// TIA Portal project "ExamenTIA" (V15)

(* hardware
DEVICE "S7-1200 station_1"  S7-1200 Station
   slot 0: "Rack_0"  S7-1200 Rack  Rack  V1.0
   slot 1: "PLC_1"  CPU 1214C AC/DC/Rly  6ES7 214-1BG40-0XB0  V4.2
*)

// ===== PLC "PLC_1"  CPU 1214C AC/DC/Rly =====

VAR_GLOBAL   // PLC tag table "Tabla de variables estándar"
   "Clock_Byte" AT %MB0 : Byte;
   "Clock_10Hz" AT %M0.0 : Bool;
   "Clock_5Hz" AT %M0.1 : Bool;
   "Clock_2.5Hz" AT %M0.2 : Bool;
   "Clock_2Hz" AT %M0.3 : Bool;
   "Clock_1.25Hz" AT %M0.4 : Bool;
   "Clock_1Hz" AT %M0.5 : Bool;
   "Clock_0.625Hz" AT %M0.6 : Bool;
   "Clock_0.5Hz" AT %M0.7 : Bool;
   "S_Abajo" AT %I0.0 : Bool;
   "S_Arriba" AT %I0.1 : Bool;
   "S_Peso" AT %I0.2 : Bool;
   "Seta" AT %I0.3 : Bool;
   "Auto" AT %I0.4 : Bool;
   "Manu" AT %I0.5 : Bool;
   "M_Alante" AT %I0.6 : Bool;
   "M_Atras" AT %I0.7 : Bool;
   "Paro" AT %I1.0 : Bool;
   "Rearme" AT %I1.1 : Bool;
   "Motor_Alante" AT %Q0.0 : Bool;
   "Motor_Atras" AT %Q0.1 : Bool;
   "L_Alante" AT %Q0.2 : Bool;
   "L_Paro" AT %Q0.3 : Bool;
   "L_ParoE" AT %Q0.4 : Bool;
   "L_Atras" AT %Q0.5 : Bool;
   "L_Sobrecarga" AT %Q0.6 : Bool;
   "FlancoP" AT %M10.0 : Bool;
   "Aux_seta" AT %M10.1 : Bool;
   "Aux_sobrecarga" AT %M10.2 : Bool;
   "FlancoN" AT %M10.3 : Bool;
   "Aux1" AT %M10.4 : Bool;
END_VAR

// folder: System blocks/Program resources

DATA_BLOCK "IEC_Timer_0_DB"   // DB1
{ S7_Optimized_Access := 'TRUE' }
AUTHOR : Simatic
FAMILY : IEC
NAME : IEC_TMR
VERSION : 1.0
// stored: InstanceOfName IEC_TIMER
"IEC_TIMER"
BEGIN
END_DATA_BLOCK

// folder: (top level)

FUNCTION "Automático" : Void   // FC1, LAD
{ S7_Optimized_Access := 'TRUE' }
VERSION : 0.1
   VAR_TEMP   // added for the SCL form of the ladder/FBD networks
      _w1 : Bool;
   END_VAR
BEGIN

REGION Network 1
   // Cuando el sensor de abajo detecta a peso activa la rampa y reinicia el temporizador de paro
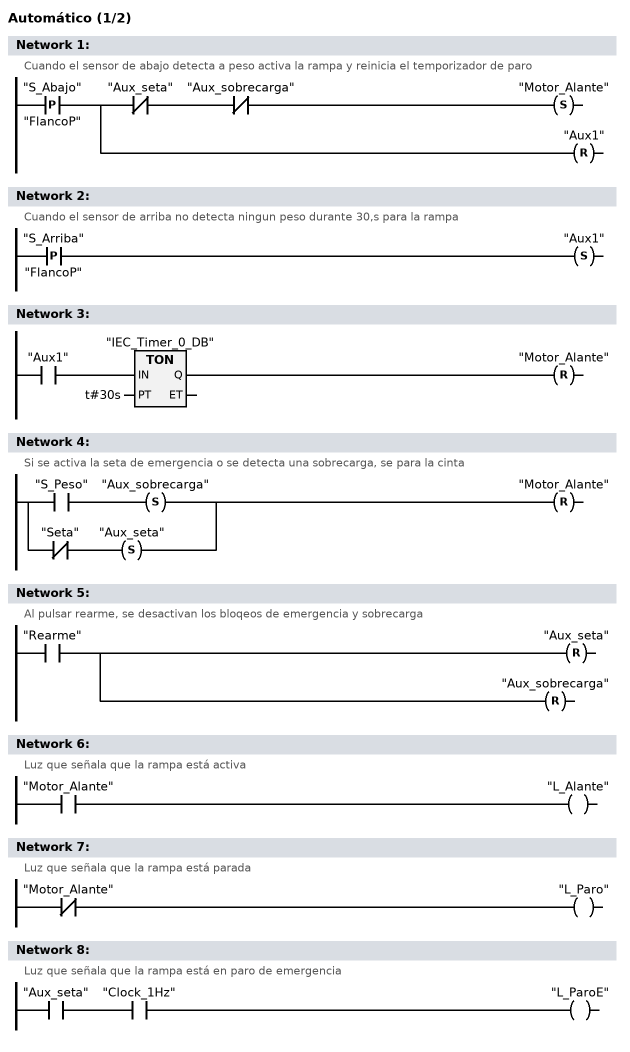
   RUNG wire#powerrail
      P_Contact(operand := "S_Abajo", bit := "FlancoP")
      wire#w1
      I_Contact( "Aux_seta" )
      I_Contact( "Aux_sobrecarga" )
      S_Coil( "Motor_Alante" )
   END_RUNG
   RUNG wire#w1
      R_Coil( "Aux1" )
   END_RUNG
   // the same network as SCL:
   #_w1 := "S_Abajo" AND NOT "FlancoP";   // rising edge of "S_Abajo"
   "FlancoP" := "S_Abajo";
   IF #_w1 AND NOT "Aux_seta" AND NOT "Aux_sobrecarga" THEN "Motor_Alante" := TRUE; END_IF;
   IF #_w1 THEN "Aux1" := FALSE; END_IF;
END_REGION

REGION Network 2
   // Cuando el sensor de arriba no detecta ningun peso durante 30,s para la rampa
   RUNG wire#powerrail
      P_Contact(operand := "S_Arriba", bit := "FlancoP")
      S_Coil( "Aux1" )
   END_RUNG
   // the same network as SCL:
   #_w1 := "S_Arriba" AND NOT "FlancoP";   // rising edge of "S_Arriba"
   "FlancoP" := "S_Arriba";
   IF #_w1 THEN "Aux1" := TRUE; END_IF;
END_REGION

REGION Network 3
   "IEC_Timer_0_DB".TON(IN := "Aux1", PT := t#30s);
   IF "IEC_Timer_0_DB".Q THEN "Motor_Alante" := FALSE; END_IF;
END_REGION

REGION Network 4
   // Si se activa la seta de emergencia o se detecta una sobrecarga, se para la cinta
   RUNG wire#powerrail
      Contact( "S_Peso" )
      S_Coil( "Aux_sobrecarga" )
      wire#w1
      R_Coil( "Motor_Alante" )
   END_RUNG
   RUNG wire#powerrail
      I_Contact( "Seta" )
      S_Coil( "Aux_seta" )
   END_RUNG wire#w1
   // the same network as SCL:
   IF "S_Peso" THEN "Aux_sobrecarga" := TRUE; END_IF;
   IF NOT "Seta" THEN "Aux_seta" := TRUE; END_IF;
   IF "S_Peso" OR NOT "Seta" THEN "Motor_Alante" := FALSE; END_IF;
END_REGION

REGION Network 5
   // Al pulsar rearme, se desactivan los bloqeos de emergencia y sobrecarga
   RUNG wire#powerrail
      Contact( "Rearme" )
      wire#w1
      R_Coil( "Aux_seta" )
   END_RUNG
   RUNG wire#w1
      R_Coil( "Aux_sobrecarga" )
   END_RUNG
   // the same network as SCL:
   IF "Rearme" THEN
       "Aux_seta" := FALSE;
       "Aux_sobrecarga" := FALSE;
   END_IF;
END_REGION

REGION Network 6
   // Luz que señala que la rampa está activa
   RUNG wire#powerrail
      Contact( "Motor_Alante" )
      Coil( "L_Alante" )
   END_RUNG
   // the same network as SCL:
   "L_Alante" := "Motor_Alante";
END_REGION

REGION Network 7
   // Luz que señala que la rampa está parada
   RUNG wire#powerrail
      I_Contact( "Motor_Alante" )
      Coil( "L_Paro" )
   END_RUNG
   // the same network as SCL:
   "L_Paro" := NOT "Motor_Alante";
END_REGION

REGION Network 8
   // Luz que señala que la rampa está en paro de emergencia
   RUNG wire#powerrail
      Contact( "Aux_seta" )
      Contact( "Clock_1Hz" )
      Coil( "L_ParoE" )
   END_RUNG
   // the same network as SCL:
   "L_ParoE" := "Aux_seta" AND "Clock_1Hz";
END_REGION

REGION Network 9
   // Luz que señala que la rampa está en paro por sobrecarga
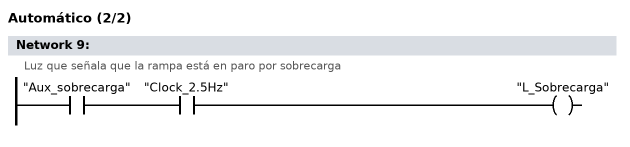
   RUNG wire#powerrail
      Contact( "Aux_sobrecarga" )
      Contact( "Clock_2.5Hz" )
      Coil( "L_Sobrecarga" )
   END_RUNG
   // the same network as SCL:
   "L_Sobrecarga" := "Aux_sobrecarga" AND "Clock_2.5Hz";
END_REGION
END_FUNCTION

FUNCTION "Manual" : Void   // FC2, LAD
{ S7_Optimized_Access := 'TRUE' }
VERSION : 0.1
BEGIN

REGION Network 1
   // Activa la rampa hacia arriba
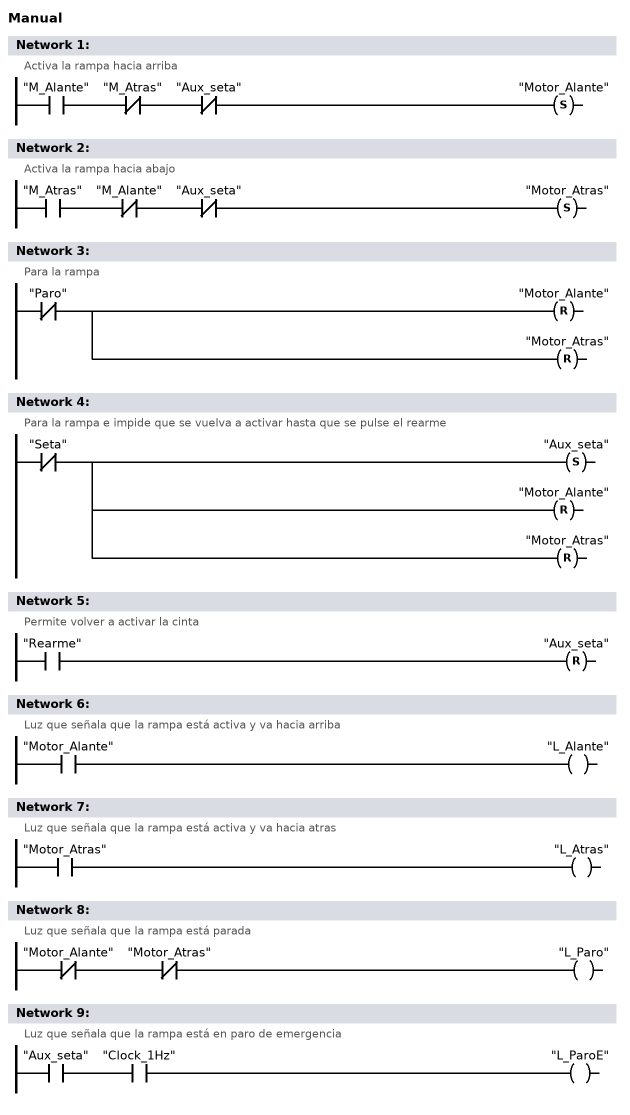
   RUNG wire#powerrail
      Contact( "M_Alante" )
      I_Contact( "M_Atras" )
      I_Contact( "Aux_seta" )
      S_Coil( "Motor_Alante" )
   END_RUNG
   // the same network as SCL:
   IF "M_Alante" AND NOT "M_Atras" AND NOT "Aux_seta" THEN "Motor_Alante" := TRUE; END_IF;
END_REGION

REGION Network 2
   // Activa la rampa hacia abajo
   RUNG wire#powerrail
      Contact( "M_Atras" )
      I_Contact( "M_Alante" )
      I_Contact( "Aux_seta" )
      S_Coil( "Motor_Atras" )
   END_RUNG
   // the same network as SCL:
   IF "M_Atras" AND NOT "M_Alante" AND NOT "Aux_seta" THEN "Motor_Atras" := TRUE; END_IF;
END_REGION

REGION Network 3
   // Para la rampa
   RUNG wire#powerrail
      I_Contact( "Paro" )
      wire#w1
      R_Coil( "Motor_Alante" )
   END_RUNG
   RUNG wire#w1
      R_Coil( "Motor_Atras" )
   END_RUNG
   // the same network as SCL:
   IF NOT "Paro" THEN
       "Motor_Alante" := FALSE;
       "Motor_Atras" := FALSE;
   END_IF;
END_REGION

REGION Network 4
   // Para la rampa e impide que se vuelva a activar hasta que se pulse el rearme
   RUNG wire#powerrail
      I_Contact( "Seta" )
      wire#w1
      S_Coil( "Aux_seta" )
   END_RUNG
   RUNG wire#w1
      R_Coil( "Motor_Alante" )
   END_RUNG
   RUNG wire#w1
      R_Coil( "Motor_Atras" )
   END_RUNG
   // the same network as SCL:
   IF NOT "Seta" THEN
       "Aux_seta" := TRUE;
       "Motor_Alante" := FALSE;
       "Motor_Atras" := FALSE;
   END_IF;
END_REGION

REGION Network 5
   // Permite volver a activar la cinta
   RUNG wire#powerrail
      Contact( "Rearme" )
      R_Coil( "Aux_seta" )
   END_RUNG
   // the same network as SCL:
   IF "Rearme" THEN "Aux_seta" := FALSE; END_IF;
END_REGION

REGION Network 6
   // Luz que señala que la rampa está activa y va hacia arriba
   RUNG wire#powerrail
      Contact( "Motor_Alante" )
      Coil( "L_Alante" )
   END_RUNG
   // the same network as SCL:
   "L_Alante" := "Motor_Alante";
END_REGION

REGION Network 7
   // Luz que señala que la rampa está activa y va hacia atras
   RUNG wire#powerrail
      Contact( "Motor_Atras" )
      Coil( "L_Atras" )
   END_RUNG
   // the same network as SCL:
   "L_Atras" := "Motor_Atras";
END_REGION

REGION Network 8
   // Luz que señala que la rampa está parada
   RUNG wire#powerrail
      I_Contact( "Motor_Alante" )
      I_Contact( "Motor_Atras" )
      Coil( "L_Paro" )
   END_RUNG
   // the same network as SCL:
   "L_Paro" := NOT "Motor_Alante" AND NOT "Motor_Atras";
END_REGION

REGION Network 9
   // Luz que señala que la rampa está en paro de emergencia
   RUNG wire#powerrail
      Contact( "Aux_seta" )
      Contact( "Clock_1Hz" )
      Coil( "L_ParoE" )
   END_RUNG
   // the same network as SCL:
   "L_ParoE" := "Aux_seta" AND "Clock_1Hz";
END_REGION
END_FUNCTION

ORGANIZATION_BLOCK "Main"   // OB1, LAD, ProgramCycle
TITLE = "Main Program Sweep (Cycle)"
{ S7_Optimized_Access := 'TRUE' }
VERSION : 0.1
   VAR_INPUT
      Initial_Call : Bool;   // Initial call of this OB
      Remanence : Bool;   // =True, if remanent data are available
   END_VAR
   VAR_TEMP   // added for the SCL form of the ladder/FBD networks
      _w1 : Bool;
      _w2 : Bool;
   END_VAR
BEGIN

REGION Network 1
   // Selector está en la posición de automatico, y entra en la subrrutina correspondiente
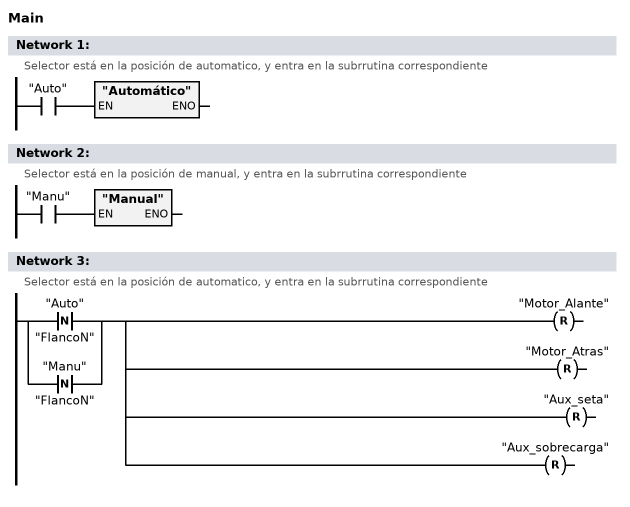
   RUNG wire#powerrail
      Contact( "Auto" )
      "Automático"()
   END_RUNG
   // the same network as SCL:
   IF "Auto" THEN "Automático"(); END_IF;
END_REGION

REGION Network 2
   // Selector está en la posición de manual, y entra en la subrrutina correspondiente
   RUNG wire#powerrail
      Contact( "Manu" )
      "Manual"()
   END_RUNG
   // the same network as SCL:
   IF "Manu" THEN "Manual"(); END_IF;
END_REGION

REGION Network 3
   // Selector está en la posición de automatico, y entra en la subrrutina correspondiente
   RUNG wire#powerrail
      N_Contact(operand := "Auto", bit := "FlancoN")
      wire#w1
      R_Coil( "Motor_Alante" )
   END_RUNG
   RUNG wire#powerrail
      N_Contact(operand := "Manu", bit := "FlancoN")
   END_RUNG wire#w1
   RUNG wire#w1
      R_Coil( "Motor_Atras" )
   END_RUNG
   RUNG wire#w1
      R_Coil( "Aux_seta" )
   END_RUNG
   RUNG wire#w1
      R_Coil( "Aux_sobrecarga" )
   END_RUNG
   // the same network as SCL:
   #_w1 := NOT "Auto" AND "FlancoN";   // falling edge of "Auto"
   "FlancoN" := "Auto";
   #_w2 := NOT "Manu" AND "FlancoN";   // falling edge of "Manu"
   "FlancoN" := "Manu";
   IF #_w1 OR #_w2 THEN
       "Motor_Alante" := FALSE;
       "Motor_Atras" := FALSE;
       "Aux_seta" := FALSE;
       "Aux_sobrecarga" := FALSE;
   END_IF;
END_REGION
END_ORGANIZATION_BLOCK